{attribute 'qualified_only'}
VAR_GLOBAL
	FilterWheel_AxisRef:		AXIS_REF;
END_VAR

(* stored: Version 1.1.0.1, ProductVersion 3.1.4024.0
   GVL GVL_FilterWheel: Id {3db1272d-8c2a-4997-9634-91e0f675134e} *)
